// SIMATIC STEP 7 (V5.x) project HW8 - Problem 2
// CPU: CPU 314C-2 DP
// station: Hardware
// station: SIMATIC 300(1)
// station: P_ADR_BUS
// program: S7 Program(2)

ORGANIZATION_BLOCK OB 1
TITLE = "Main Program Sweep (Cycle)"
//HW8 - plc - Problem 2 
VERSION : 0.1
VAR_TEMP
  OB1_EV_CLASS : BYTE ;	//Bits 0-3 = 1 (Coming event), Bits 4-7 = 1 (Event class 1)
  OB1_SCAN_1 : BYTE ;	//1 (Cold restart scan 1 of OB 1), 3 (Scan 2-n of OB 1)
  OB1_PRIORITY : BYTE ;	//Priority of OB Execution
  OB1_OB_NUMBR : BYTE ;	//1 (Organization block 1, OB1)
  OB1_RESERVED_1 : BYTE ;	//Reserved for system
  OB1_RESERVED_2 : BYTE ;	//Reserved for system
  OB1_PREV_CYCLE : INT ;	//Cycle time of previous OB1 scan (milliseconds)
  OB1_MIN_CYCLE : INT ;	//Minimum cycle time of OB1 (milliseconds)
  OB1_MAX_CYCLE : INT ;	//Maximum cycle time of OB1 (milliseconds)
  OB1_DATE_TIME : DATE_AND_TIME ;	//Date and time OB1 started
END_VAR
BEGIN
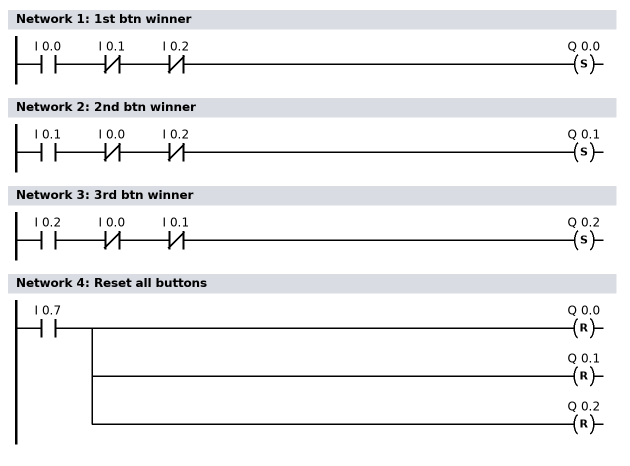
NETWORK
TITLE = 1st btn winner
      A     I 0.0;
      AN    I 0.1;
      AN    I 0.2;
      S     Q 0.0;
NETWORK
TITLE = 2nd btn winner
      A     I 0.1;
      AN    I 0.0;
      AN    I 0.2;
      S     Q 0.1;
NETWORK
TITLE = 3rd btn winner
      A     I 0.2;
      AN    I 0.0;
      AN    I 0.1;
      S     Q 0.2;
NETWORK
TITLE = Reset all buttons
      A     I 0.7;
      R     Q 0.0;
      R     Q 0.1;
      R     Q 0.2;
END_ORGANIZATION_BLOCK
